FUNCTION_BLOCK FB_ErrorManager
VAR
	ErrorList : ARRAY[0..20] OF ST_Error;
	index : INT;
END_VAR

METHOD ClearError : BOOL
VAR_INPUT
END_VAR
index := 0;
MEMSET(ADR(ErrorList), 0, SIZEOF(ErrorList));
END_METHOD

METHOD RaiseError : BOOL
VAR_INPUT
	ErrorCode : UINT;
	ErrorMsg : STRING;
END_VAR
VAR
	i : INT;
END_VAR
IF index < 0 OR index >= 20 THEN
	RaiseError := FALSE;
	RETURN;
END_IF

FOR i := 0 TO 20 BY 1 DO
	IF ErrorList[i].ErrorCode = ErrorCode THEN
		RaiseError := FALSE;
		RETURN;
	END_IF
END_FOR

ErrorList[index].ErrorCode := ErrorCode;
ErrorList[index].ErrorMessage := ErrorMsg;
index := index + 1;
RaiseError := TRUE;
END_METHOD

END_FUNCTION_BLOCK

(* stored: Version 1.1.0.1, ProductVersion 3.1.4024.13
   POU FB_ErrorManager: Id {6c983e80-6740-4860-b674-7fdc2a53239f}, SpecialFunc None
   Method ClearError: Id {a0d1a433-cdb8-45e9-ad91-9cac1ac35ab4}
   Method RaiseError: Id {3a15478b-ae88-4719-bba7-70e61db18687} *)
